TYPE TupleStruct_1:
    STRUCT
        field0: DINT;
        field1: DINT;
    END_STRUCT
END_TYPE

(* stored: ProductVersion 3.1.0.18, Version 1.1.0.1 *)
